// TIA Portal V20 export
TYPE "S300Manual"
// stored: Access Published, Namespace Global
   STRUCT
      GoUp : Bool;
      GoStraight : Bool;
      GoLeft : Bool;
      GoRight : Bool;
   END_STRUCT;
END_TYPE
